FUNCTION_BLOCK FB_Flasher
VAR_INPUT
		bStart: BOOL;
END_VAR
VAR_OUTPUT
	bLed: BOOL;
END_VAR
VAR
	nState: INT;
	TF1: TON;
	TF2: TON;
END_VAR



CASE nState	OF
	

	0:
		IF bStart THEN
			nState := 10;
		END_IF
		
	10:
	
		bLed	:=	TRUE;
	
		TF1(IN:=TRUE , PT:=T#500MS);
		
		IF TF1.Q THEN
			TF1(IN:=FALSE);
			nState := 20;
		END_IF
		
	20:
	
		bLed	:=	FALSE;
	
		TF2(IN:=TRUE , PT:=T#500MS);
		
		IF TF2.Q THEN
			TF2(IN:=FALSE);
			nState := 0;
		END_IF
		

END_CASE

END_FUNCTION_BLOCK

(* stored: Version 1.1.0.1, ProductVersion 3.1.4024.4
   POU FB_Flasher: Id {fd5fa9e1-16fa-43b1-bc5f-41adf27bea9c}, SpecialFunc None *)
